Staubli VAL3: setMobile.pgx

public program setMobile(string x_sItem, frame x_fFrame)
begin
  // set the frame mobile
  tTraj[x_sItem].fMoving.trsf={0,0,0,0,0,0}
  link(tTraj[x_sItem].fMoving,x_fFrame)
end
